// LS Electric XG5000 project: 동남97
// PLC NewPLC
// module base 0 slot 0: 입출력 모듈:XBC-DN/DP14E (DC 24V 입력 8점, 트랜지스터 출력 6점)

PROGRAM NewProgram (task: 스캔 프로그램)

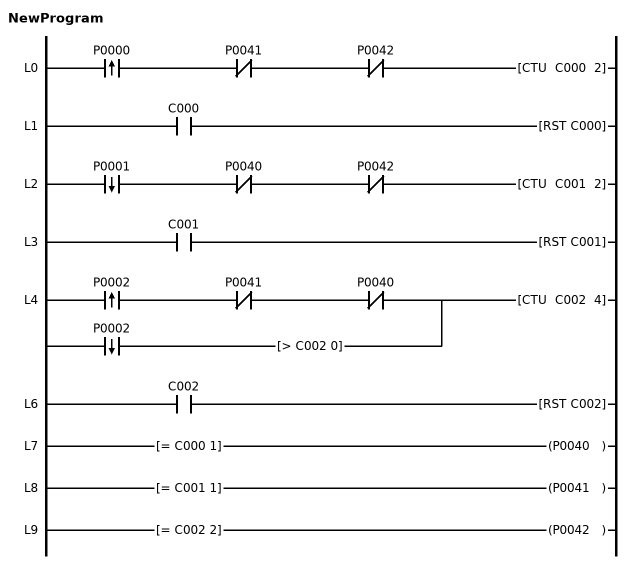
; L0
LOADP     P0000
AND NOT   P0041
AND NOT   P0042
CTU       C000 2
; L1
LOAD      C000
RST       C000
; L2
LOADN     P0001
AND NOT   P0040
AND NOT   P0042
CTU       C001 2
; L3
LOAD      C001
RST       C001
; L4
LOADP     P0002
AND NOT   P0041
AND NOT   P0040
LOADN     P0002
AND>      C002 0
OR LOAD
CTU       C002 4
; L6
LOAD      C002
RST       C002
; L7
LOAD=     C000 1
OUT       P0040
; L8
LOAD=     C001 1
OUT       P0041
; L9
LOAD=     C002 2
OUT       P0042